// Mitsubishi GX Works2 project: 3   PLC: FX3U/FX3UC

// task Task_01 (event TRUE, interval 0, priority 31): POU_01

PROGRAM POU_01
VAR
  wstep : INT;
  TON_BZ : TON;
  R_TRIG_COS_1 : R_TRIG;
  R_TRIG_COS_0 : R_TRIG;
  R_TRIG_COS_2 : R_TRIG;
  R_TRIG_THRY_ALL : R_TRIG;
  TON_SYNC : TON;
  R_TRIG_COS_PB4 : R_TRIG;
END_VAR
M99 := 
Y1 AND Y2 AND Y3 AND Y4 AND Y5 AND Y0 AND
Y10 AND Y11 AND

X1 AND X2 AND X3 AND X4 AND X0 AND
X11 AND X10 AND X12 AND
X5 AND X6 AND
X15 AND X16;

(*PB1 - X1*)						(*PL1 - Y1*)
(*PB2 - X2*)						(*PL2 - Y2*)
(*PB3 - X3*)						(*PL3 - Y3*)
(*PB4 - X4*)						(*PL4 - Y4*)
(*EMS NC - X0*)				(*PL5 - Y5*)
(*COS 1 - X11*)				(*BZ - Y0*)
(*COS 0 - X10*)				(*MC1 - Y10*)
(*COS 2 - X12*)				(*MC2 - Y11*)
(*TH-RY 1 NC - X5*)	
(*TH-RY 2 NC - X6*)
(*MC1 NO - X15*)			
(*MC2 NO - X16*)


IF M8002 THEN (*TH-RY自檢*)
	wstep := 0;
	(*開機TH-RY自檢失敗*)
	IF NOT (X5 OR X6) THEN
		wstep := 60;
	END_IF;
END_IF;

TON_SYNC(IN := (X15 XOR Y10) OR (X16 XOR Y11), PT := T#2s); (*MC無法同步*)
IF TON_SYNC.Q THEN
	wstep := 80;
END_IF;

IF wstep <> 80 THEN (*MC無法同步，則不執行*)
	IF X0 THEN (*EMS*)
		IF wstep <> 60 THEN (*TH-RY自檢失敗*)

			(*過載*)
			TON_BZ(IN := NOT (X5 AND X6), PT := T#10s); 
			
			(*TH-RY-1 跳脫*)
			IF NOT X5 THEN
				Y0 := M8013 AND NOT TON_BZ.Q;
				SET(TRUE, Y3); 		
			ELSE
				RST(TRUE, Y3);
			END_IF;
			
			(*TH-RY-2 跳脫*)
			IF NOT X6 THEN
				Y0 := M8013 AND NOT TON_BZ.Q;
				SET(TRUE, Y4); 	
			ELSE
				RST(TRUE, Y4);	
			END_IF;
			
			(*TH-RY 全部跳脫*)
			R_TRIG_THRY_ALL(_CLK := (NOT X5) AND (NOT X6));
			IF R_TRIG_THRY_ALL.Q THEN
				wstep := 50;
			END_IF;
	
			IF wstep <> 50 THEN (*如果TH-RY全部跳脫，則不執行*)
				
				(*COS選擇*)
				R_TRIG_COS_1(_CLK := X11);
				IF R_TRIG_COS_1.Q THEN
					wstep := 0;
				END_IF;
				
				R_TRIG_COS_0(_CLK := X10);
				IF R_TRIG_COS_0.Q THEN
					wstep := 1;
				END_IF;
				
				R_TRIG_COS_2(_CLK := X12);
				IF R_TRIG_COS_2.Q THEN
					wstep := 2;
				END_IF;
				
				(*水池水量不足*)
				Y5 := NOT X1;
				IF X1 THEN
					IF wstep >= 20 AND wstep < 29 THEN
						wstep := 0;
					END_IF;
					IF wstep >= 30 AND wstep < 39 THEN
						wstep := 1;
					END_IF;
				END_IF;
			END_IF;
		ELSE (*TH-RY自檢失敗*)
			wstep := 60;
		END_IF; 	
	ELSE (*EMS*)
		wstep := 70;
	END_IF;
END_IF;

CASE wstep OF
	0: 
		ZRST(TRUE, Y0, Y17);
		IF NOT X1 THEN
			wstep := 20;
		END_IF;
	1:
		ZRST(TRUE, Y0, Y17);
		IF NOT X1 THEN
			wstep := 30;
		END_IF;
	2:
		ZRST(TRUE, Y0, Y17);
		IF NOT X1 THEN
			wstep := 40;
		END_IF;
		
	20: (*COS 1*)
		RST(TRUE, Y11);
		RST(TRUE, Y2);	
		
		IF X2 THEN
			SET(TRUE, Y10);
			SET(TRUE, Y1);
		END_IF;		
		IF ((NOT X2) AND Y10) OR (NOT X5) THEN
				wstep := 21;
		END_IF;	
	21: 
		RST(TRUE, Y10);
		RST(TRUE, Y1);
		
		IF X2 THEN
			SET(TRUE, Y11);
			SET(TRUE, Y2);
		END_IF;
		IF ((NOT X2) AND Y11) OR (NOT X6) THEN
				wstep := 20;
		END_IF;

	30: (*COS 0*)
		RST(TRUE, Y11);
		RST(TRUE, Y2);		
		R_TRIG_COS_PB4(_CLK := X4);
		IF R_TRIG_COS_PB4.Q OR (NOT X5) THEN
			wstep := 31;
		END_IF;
	31:
		SET(TRUE, Y10);
		SET(TRUE, Y1);
		R_TRIG_COS_PB4(_CLK := X4);
		IF R_TRIG_COS_PB4.Q OR (NOT X5) THEN
			wstep := 32;
		END_IF;		
	32:
		RST(TRUE, Y10);
		RST(TRUE, Y1);		
		R_TRIG_COS_PB4(_CLK := X4);
		IF R_TRIG_COS_PB4.Q OR (NOT X6) THEN
			wstep := 33;
		END_IF;
	33:
		SET(TRUE, Y11);
		SET(TRUE, Y2);
		R_TRIG_COS_PB4(_CLK := X4);
		IF R_TRIG_COS_PB4.Q OR (NOT X6) THEN
			wstep := 30;
		END_IF;
		 
	40: (*COS 2*)
		IF X1 THEN
			wstep := 2;
		END_IF;		
	
		IF X2 THEN		
			
			(*第一機*)
			IF X5 THEN
				SET(TRUE, Y10);	
				SET(TRUE, Y1);
			ELSE
				RST(TRUE, Y10);
				RST(TRUE, Y1);
			END_IF;
			
			(*第二機*)
			IF X6 THEN
				SET(TRUE, Y11);
				SET(TRUE, Y2);
			ELSE
				RST(TRUE, Y11);
				RST(TRUE, Y2);
			END_IF;
		ELSE
			RST(TRUE, Y10);
			RST(TRUE, Y11);
			RST(TRUE, Y1);
			RST(TRUE, Y2);			
		END_IF;
	
	50: (*TH-RY全部跳脫*)
		ZRST(TRUE, Y0, Y17);
		SET(TRUE, Y3);
		SET(TRUE, Y4);
		Y0 := M8013;
		IF X3 THEN
			wstep := 51;
		END_IF;
	51:
		IF X5 AND X6 THEN
			wstep := 52;
		END_IF;	
	52:
		IF X11 THEN
			wstep := 0;
		END_IF;
		IF X10 THEN
			wstep := 1;
		END_IF;
		IF X12 THEN
			wstep := 2;
		END_IF;
	
	60: (*TH-RY開機自檢失敗*)
		Y3 := M8013 AND (NOT X5);
		Y4 := M8013 AND (NOT X6);
		IF X5 AND X6 THEN
			IF X11 THEN
				wstep := 0;
			END_IF;
			IF X10 THEN
				wstep := 1;
			END_IF;
			IF X12 THEN
				wstep := 2;
			END_IF;
		END_IF;
			
	70: (*EMS*)
		ZRST(TRUE, Y0, Y17);
		
	80: (*MC無法同步*)
		ZRST(TRUE, Y0, Y17);
		
END_CASE;
END_PROGRAM
